// SIMATIC STEP 7 (V5.x) project TEMA 13 EJERCICIO 35
// CPU: CPU313 C-2 DP(1)
// station: P_ADR_BUS
// station: Hardware
// station: Equipo SIMATIC 300
// program: Programa S7(1)

SYMBOL_TABLE
"Cycle Execution"	OB 1	OB 1
END_SYMBOL_TABLE
